Fanuc KAREL source: ka00079.KL

-- PROVISIONAL review KL for V770-1; original PC SHA256 fba543c86008f12358e8da7fb0eb85d2cde2c5d0e0915c5a3881d0477bb2b1a1
-- Incomplete behavior may be omitted. Consult companion uncertainty JSON. Do not deploy.
PROGRAM KA00079
%NOLOCKGROUP
-- UNRESOLVED_DECL SRC type=000106
-- UNRESOLVED_DECL DST type=000106
BEGIN
  -- UNRESOLVED_PC offsets 5-20; opcodes 2E,22,32,35
  -- UNRESOLVED_PC offsets 25-40; opcodes 49,4A
  -- UNRESOLVED_PC offsets 45-49; opcodes 7F
END KA00079
